// TwinCAT 3 PLC project Untitled1
// ProgramVersion: 3.1.4026.10
// libraries:
//   Tc2_Standard, * (Beckhoff Automation GmbH)
//   Tc2_System, * (Beckhoff Automation GmbH)
//   Tc2_Utilities, * (Beckhoff Automation GmbH)
//   Tc3_IotBase, * (Beckhoff Automation GmbH)
// project tree:
//   / PlcTask.TcTTO
//   POUs/ MAIN.TcPOU
// real-time tasks:
//   TASK PlcTask: cycle T#10ms, priority 20, ADS port 350
// I/O:
//   DEVICE Device 1 (EtherCAT), AmsNetId 192.168.1.1.2.1
//     Term 1 (EK1200) [EK1200-5000 EtherCAT Power supply (2A E-Bus)]
//       Term 2 (EL1859) [EL1859 8Ch. Dig. Input 24V, 3ms, 8Ch. Dig. Output 24V, 0.5A]
//       Term 3 (EL1859) [EL1859 8Ch. Dig. Input 24V, 3ms, 8Ch. Dig. Output 24V, 0.5A]
//       Term 4 (EL3255) [EL3255 5Ch. potentiometer measurement with sensor supply]
//       Term 5 (EL3214-0090) [EL3214-0090 4Ch. Ana. Input PT100 (RTD), TwinSAFE SC]
//       Term 6 (EL5151) [EL5151 1Ch. Inc. Encoder]
//       Term 7 (EL1904) [EL1904, 4 Ch. Safety Input 24V, TwinSAFE]
//         modules: Module 1 (FSOES)
//       Term 8 (EL2904) [EL2904, 4 Ch. Safety Output 24V, 0.5A, TwinSAFE]
//         modules: Module 1 (FSOES), Module 2 (DO)
//       Term 9 (EL6910) [EL6910, TwinSAFE PLC]
//       Term 10 (EL9110) [EL9110 Power Supplier with LED (24V, Diagnostics)]
//       Term 11 (EL7201-9014) [EL7201-9014 1Ch. MDP742 Servo motor output stage with OCT (50V, 2.8A RMS) and STO input]
//       Term 12 (EL9011) [EL9011 End Terminal]
//   DEVICE CX51662_MQTT
//     Box 15 (Publisher)
//     Box 13 (Subscriber)
// variable links:
//   Untitled1/Untitled1 Instance <-> CX51662_MQTT/Box 13 (Subscriber)
//     PlcTask Inputs/MAIN.iEL3255_Sub <-> EL3255/Inputs/VarData
//   Untitled1/Untitled1 Instance <-> CX51662_MQTT/Box 15 (Publisher)
//     PlcTask Outputs/MAIN.iEL3255_Pub <-> EL3255/Outputs/VarData
//   Untitled1/Untitled1 Instance <-> Device 1 (EtherCAT)/Term 1 (EK1200)/Term 4 (EL3255)
//     PlcTask Inputs/MAIN.iEL3255_In <-> AI Standard Channel 1/Value

CONFIGURATION Untitled1
    RESOURCE PLC ON TwinCAT3
        TASK PlcTask(INTERVAL := T#10ms, PRIORITY := 20);
        PROGRAM MAIN WITH PlcTask : MAIN;
    END_RESOURCE
END_CONFIGURATION

// ---- POUs/MAIN.TcPOU
PROGRAM MAIN
VAR
	 fbMqttClient   : FB_IotMqttClient;
    bSetParameter   : BOOL := TRUE;
    bConnect        : BOOL := FALSE;
	  (* published message *)
 	sTopicPub   	: STRING(255) := 'TwinCAT_CX5166C2';
    sPayloadPub 	: STRING(255);
    fbTimer 		: TON := (PT:=T#1S);
    iCount 			: UDINT;
	  (* received message *)
    bSubscribed    	: BOOL;
    sTopicSub      	: STRING(255) := 'TwinCAT_CX5166C2';
    {attribute 'TcEncoding':='UTF-8'}
    sTopicRcv      	: STRING(255);
    {attribute 'TcEncoding':='UTF-8'}
    sPayloadRcv    	: STRING(255);
    fbMessageQueue 	: FB_IotMqttMessageQueue;
    fbMessage      	: FB_IotMqttMessage;
	state 			: INT;
	
	iEL3255_In	AT %I*	: INT;
	iEL3255_Pub	AT %Q*	: INT;
	iEL3255_Sub	AT %I*	: INT;
END_VAR

iEL3255_Pub := iEL3255_In;
//State machine
CASE state OF
	10:
		IF bSetParameter THEN
			bSetParameter               := FALSE;
			fbMqttClient.sHostName      := '169.254.135.73';
			fbMqttClient.nHostPort      := 1883;
			fbMqttClient.ipMessageQueue := fbMessageQueue;
			bSetParameter := FALSE;
		END_IF
		bConnect:=True;
		IF fbMqttClient.bConnected THEN
			state := 20;
		END_IF
	20:
	IF fbMessageQueue.nQueuedMessages > 0 THEN
  	  	IF fbMessageQueue.Dequeue(fbMessage:=fbMessage) THEN
			fbMessage.GetTopic(pTopic:=ADR(sTopicRcv), nTopicSize:=SIZEOF(sTopicRcv) );
			fbMessage.GetPayload(pPayload:=ADR(sPayloadRcv), nPayloadSize:=SIZEOF(sPayloadRcv), bSetNullTermination:=FALSE);
		END_IF
	END_IF
	
	IF NOT bSubscribed THEN
		bSubscribed := fbMqttClient.Subscribe(sTopic:=sTopicSub, eQoS:=TcIotMqttQos.AtMostOnceDelivery);
	END_IF
    fbTimer(IN:=TRUE);
    IF fbTimer.Q THEN // publish new payload every second
        fbTimer(IN:=FALSE);
        iCount := iCount + 1;
        sPayloadPub := CONCAT('MyMessage', TO_STRING(iCount));
        fbMqttClient.Publish(sTopic:= sTopicPub,
					pPayload:= ADR(sPayloadPub), 
					nPayloadSize:= LEN2(ADR(sPayloadPub))+1, 
					eQoS:= TcIotMqttQos.AtMostOnceDelivery, 
					bRetain:= FALSE, 
					bQueue:= FALSE );
    END_IF
END_CASE
fbMqttClient.Execute(bConnect:= bConnect);

END_PROGRAM
